TYPE ST_RECORD :
STRUCT
	listRecordData:		ARRAY[0..2999] OF ST_RECORD_DATA;
END_STRUCT
END_TYPE

(* stored: Version 1.1.0.1, ProductVersion 3.1.4024.12
   DUT ST_RECORD: Id {d541417c-59f7-4e01-b634-3c888cf8240d} *)
